FUNCTION_BLOCK FB_Observer_REAL EXTENDS FB_AbstractObserver
VAR
    _fVal:              REAL;
END_VAR

METHOD FB_init : BOOL
VAR_INPUT
	bInitRetains : BOOL; // if TRUE, the retain variables are initialized (warm start / cold start)
	bInCopyCode : BOOL;  // if TRUE, the instance afterwards gets moved into the copy code (online change)
END_VAR
THIS^._nTypeClass := __SYSTEM.TYPE_CLASS.TYPE_REAL;
THIS^._pVal := ADR(THIS^._fVal);
THIS^._nSize := SIZEOF(THIS^._fVal);
END_METHOD

PROPERTY fValue32 : REAL
GET
fValue32 := THIS^._fVal;
END_GET
END_PROPERTY

END_FUNCTION_BLOCK

(* stored: Version 1.1.0.1, ProductVersion 3.1.4024.12
   POU FB_Observer_REAL: Id {d1c7af26-f07e-42b0-992b-a1ffff6d7b81}, SpecialFunc None
   Method FB_init: Id {dcd4bf04-a6c5-0c5a-0813-1d36612f0369}
   Property fValue32: Id {c642b59a-6e55-4cd0-8595-4cc6183b71c8}
   Get Get: Id {3fab4433-5f59-4791-9081-0075f9ea3bcd} *)
